// TIA Portal V17 export
// export: Created 2023-12-29T10:44:22.8737876Z, ExportSetting None, DisplayName Totally Integrated Automation Portal, DisplayVersion V17 Update 4, DisplayName TIA Portal Openness, DisplayVersion V17 Update 4, DisplayName TIA Portal Version Control Interface, DisplayVersion V17, DisplayName STEP 7 Professional, DisplayVersion V17 Update 4, DisplayName STEP 7 Safety, DisplayVersion V17, DisplayName WinCC Advanced / Unified PC, DisplayVersion V17 Update 4
FUNCTION "FC_AIn2oo3" : Void   // FC555, LAD
{ S7_Optimized_Access := 'FALSE' }
// AnalogInput2oo3
// stored: AutoNumber false, SetENOAutomatically false
BEGIN
END_FUNCTION
